PROGRAM PRG_VFS
VAR
END_VAR

//Fast Shutter Valve
//H1
TV2K3_VFS_01(
    i_xVeto_Enable:=False,
    i_xPMPS_OK:= TRUE,
    i_xExt_OK:= TRUE,
    i_sDevName:= 'TV2K3:VFS:01',
    io_fbFFHWO:= GVL_PMPS.g_FastFaultOutput2
    );

END_PROGRAM

(* stored: Version 1.1.0.1, ProductVersion 3.1.4024.12
   POU PRG_VFS: Id {44a96bd7-db4e-4158-b32e-0c3edb6ec23b}, SpecialFunc None *)
